(* Logix 5000 project; controller Arrow3 vendor 1 type 14 code 235 rev 36.11; software revision 36.00; part 3 of 3 *)

PROGRAM SafetyProgram   (* main routine MainRoutine, safety *)

ROUTINE MainRoutine   (* ladder *)
END_ROUTINE
END_PROGRAM
